PROGRAM MAIN
VAR
	bEntrada01	:	BOOL;
	bEntrada02	:	BOOL;
	bSalida01	:	BOOL;
	bSalida02	:	BOOL;	
END_VAR


bEntrada01 := bEntrada02;
bSalida01 := bSalida02;

END_PROGRAM

(* stored: Version 1.1.0.1, ProductVersion 3.1.4024.13
   POU MAIN: Id {723e5577-28d8-48dc-a83c-01152d265357}, SpecialFunc None *)
